INTERFACE I_Dictionary

END_INTERFACE

(* stored: Version 1.1.0.1
   Itf I_Dictionary: Id {fb4ff7d0-fb23-0fc0-23a7-39f8a7884151} *)
